PROGRAM Step_Log_Clear
VAR
	db_fb_PLCDBCmdEvt : FB_PLCDBCmdEvt(sNetID:= '', tTimeout:= T#5S );
	
	_stPara		: ARRAY [0..3] OF ST_ExpParameter;
	
	_SqlCommand : STRING(1024);
	
	_extrasstr : STRING(255);
	
	_fbJson      : FB_JsonSaxWriter;
	Clear_date: LINT;
END_VAR

Clear_date := TO_LINT(F_GetSystemTime());

// SQL命令
_SqlCommand := 

'DELETE 
	INTO program_running_log 
		(program_name, step_number, created_at, detail_data)
	VALUES
		({program_name}, {step_number}, to_timestamp(({created_at} - 116444736000000000) / 10000000.0), {detail_data}::jsonb);
';


db_fb_PLCDBCmdEvt.Execute(
	hDBID := 3,
	pExpression := ADR(_SqlCommand),			// SQL 命令 ex. SELECT * FROM PlcTest.newtable WHERE ID = {ID}  
	cbExpression := SIZEOF(_SqlCommand),		// SQL 命令字串的長度
	pData:= 0,		// 帶入的參數值
	cbData:= 0,//itmp, 	// 帶入的參數值大小
	pParameter:= 0, 				// 帶入的參數類型設定  ex.上面命令內的 {ID} 類型設定
	cbParameter:= 0,			// 帶入的參數類型設定的大小
)

{attribute 'suppress_wrn_C0410'}
PROPERTY fbJson : REFERENCE TO FB_JsonSaxWriter
GET
fbJson REF= _fbJson;
END_GET
END_PROPERTY

METHOD JsonOutput : BOOL
VAR_INPUT
END_VAR
fbJson.EndObject();
_extrasstr := fbJson.GetDocument();
fbJson.ResetDocument();
END_METHOD

END_PROGRAM

(* stored: Version 1.1.0.1, ProductVersion 3.1.4026.13
   POU Step_Log_Clear: Id {9f3db44a-1879-4a93-ada6-f6fd1c5e22d1}, SpecialFunc None
   Property fbJson: Id {22b63b51-49bd-4cb3-aee3-95cf126aa71f}
   Get Get: Id {45dc1dab-0b7c-47d5-91e0-f88e56ddf519}
   Method JsonOutput: Id {8e99a240-a291-4b5a-8e93-a0e6b6bae871} *)
